% RSLogix 500 project 2_AUTOMATIC_BOTTLE_FILLING_MACHINE.RSS, saved by version 8.30.00.16 %
PROJECT "1"    % processor: MicroLogix 1000 %

PROGRAM FILES
  LAD 2 "MAIN_PROG"  6 rungs
  LAD 3 "USER_FAULT"  1 rungs
  LAD 4 "HSC_INT"  1 rungs
  LAD 5 "STI_INT"  1 rungs
  LAD 6, 7, 8, 9, 10, 11, 12, 13, 14, 15, 16: only END

DATA FILES
  O0 OUTPUT  1 elements
  I1 INPUT  2 elements
  S2 STATUS  33 elements
  B3 BINARY  32 elements
  T4 TIMER  40 elements
  C5 COUNTER  32 elements
  R6 CONTROL  16 elements
  N7 INTEGER  105 elements

LADDER 2 "MAIN_PROG"
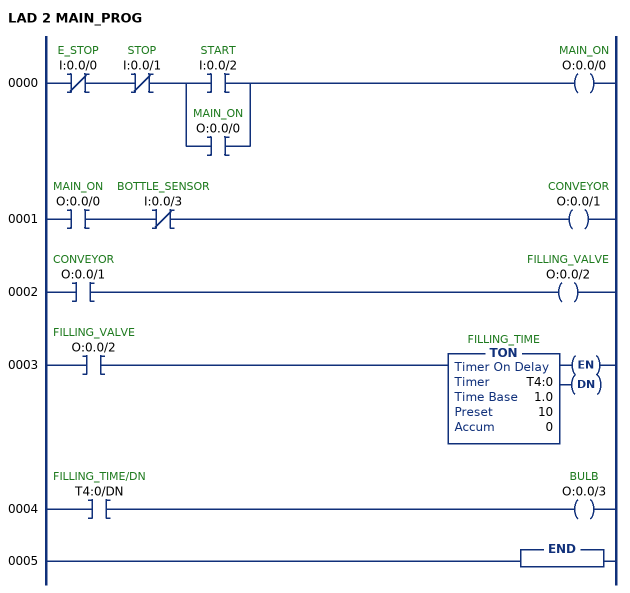
% Rung: 0 %
SOR XIO I:0.0/0 XIO I:0.0/1 BST XIC I:0.0/2 NXB XIC O:0.0/0 BND OTE O:0.0/0 EOR
%   I:0.0/0  E_STOP %
%   I:0.0/1  STOP %
%   I:0.0/2  START %
%   O:0.0/0  MAIN_ON %
% Rung: 1 %
SOR XIC O:0.0/0 XIO I:0.0/3 OTE O:0.0/1 EOR
%   O:0.0/0  MAIN_ON %
%   I:0.0/3  BOTTLE_SENSOR %
%   O:0.0/1  CONVEYOR %
% Rung: 2 %
SOR XIC O:0.0/1 OTE O:0.0/2 EOR
%   O:0.0/1  CONVEYOR %
%   O:0.0/2  FILLING_VALVE %
% Rung: 3 %
SOR XIC O:0.0/2 TON T4:0 1.0 10 0 EOR
%   O:0.0/2  FILLING_VALVE %
%   T4:0  FILLING_TIME %
% Rung: 4 %
SOR XIC T4:0/DN OTE O:0.0/3 EOR
%   T4:0  FILLING_TIME %
%   O:0.0/3  BULB %
% Rung: 5 %
SOR END EOR

DATA TABLE (non-zero values as saved)
DATA T4
% .PRE .ACC %
% T4:0 % 10 0
